# EPICS autosave request: iocBoot/ioc13bmd_pace5000/auto_settings.req
file "PACE5000_settings.req",       P=$(P), R=PC1:
